FUNCTION_BLOCK PUBLIC FINAL FB_CodedOutputStream
VAR_IN_OUT
    aBuffer : ARRAY [*] OF BYTE;
END_VAR
VAR
    stState : ST_WriterInternalState;
END_VAR

{warning 'TODO: Field codecs for FB_CodedOutputStream'}
VAR
//     fbFieldCodecInt32           : FB_FieldCodecInt32;
    fbFieldCodecUInt32          : FB_FieldCodecUInt32;
//     fbFieldCodecInt64       : FB_FieldCodecInt64;
//     fbFieldCodecSInt32      : FB_FieldCodecSInt32;
//     fbFieldCodecSInt64      : FB_FieldCodecSInt64;
//     fbFieldCodecFixed32     : FB_FieldCodecFixed32;
//     fbFieldCodecFixed64     : FB_FieldCodecFixed64;    
//     fbFieldCodecFloat       : FB_FieldCodecFloat;
//     fbFieldCodecDouble      : FB_FieldCodecDouble;
    fbFieldCodecString      : FB_FieldCodecString;
//     fbFieldCodecBytes       : FB_FieldCodecBytes;
//     fbFieldCodecBool        : FB_FieldCodecBool;
END_VAR

METHOD PUBLIC FromBuffer : HRESULT
VAR
    hr : HRESULT;
END_VAR

Reset();

hr := ValidateBuffer(aBuffer);
IF FAILED(hr) THEN
    FromBuffer := hr;
    RETURN;
END_IF

Init(aBuffer);
END_METHOD

METHOD PRIVATE Init
VAR_IN_OUT CONSTANT
    aBuffer : ARRAY [*] OF BYTE;
END_VAR
VAR
    nSize : DINT;
END_VAR

stState.nBufferPos := TO_UDINT(LOWER_BOUND(aBuffer, 1));

nSize := UPPER_BOUND(aBuffer, 1) - LOWER_BOUND(aBuffer, 1);
stState.nBufferSize := TO_UDINT(nSize);
END_METHOD

PROPERTY nSpaceLeft : UDINT
GET
nSpaceLeft := stState.nBufferSize - stState.nBufferPos;
END_GET
END_PROPERTY

METHOD PRIVATE Reset
VAR_INPUT
END_VAR

stState.bError := FALSE;
stState.eWriterErrorCode := S_OK;
stState.nBufferPos := 0;
stState.nBufferSize := 0;
END_METHOD

METHOD PRIVATE ValidateBuffer : HRESULT
VAR_IN_OUT CONSTANT
    aBuffer : ARRAY[*] OF BYTE;
END_VAR
VAR
    nSize : DINT;
END_VAR
IF LOWER_BOUND(aBuffer, 1) < 0 THEN
    ValidateBuffer := E_CodedOutputStreamErrorCode.BUFFER_LOWER_BOUND;
    RETURN;
END_IF

nSize := UPPER_BOUND(aBuffer, 1) - LOWER_BOUND(aBuffer, 1);
IF nSize = 0 OR TO_UDINT(nSize) >  Param_PB.cMaxProtobufRawBuffer THEN
    ValidateBuffer := E_CodedOutputStreamErrorCode.BUFFER_SIZE;
    RETURN;
END_IF
END_METHOD

METHOD WriteBool : HRESULT
VAR_INPUT
    bValue : BOOL;
END_VAR

WriteBool := F_WriteRawByte(aBuffer, stState, TO_BYTE(bValue));
END_METHOD

METHOD WriteBytes : HRESULT
VAR_IN_OUT CONSTANT
    aBytes  : ARRAY [*] OF BYTE;
END_VAR
VAR_INPUT
    nLength : UDINT;
END_VAR

WriteBytes := F_WriteBytes(aBuffer, stState, aBytes, nLength);
END_METHOD

METHOD WriteDouble : HRESULT
VAR_INPUT
    fValue : LREAL;
END_VAR
WriteDouble := F_WriteDouble(aBuffer, stState, fValue);
END_METHOD

METHOD WriteEnum : HRESULT
VAR_INPUT
    nValue : DINT;
END_VAR

WriteEnum := F_WriteEnum(aBuffer, stState, nValue);
END_METHOD

METHOD WriteFixed32 : HRESULT
VAR_INPUT
    nValue : UDINT;
END_VAR

WriteFixed32 := F_WriteFixed32(aBuffer, stState, nValue);
END_METHOD

METHOD WriteFixed64 : HRESULT
VAR_INPUT
    nValue : ULINT;
END_VAR

WriteFixed64 := F_WriteFixed64(aBuffer, stState, nValue);
END_METHOD

METHOD WriteFloat : HRESULT
VAR_INPUT
    fValue : REAL;
END_VAR
WriteFloat := F_WriteFloat(aBuffer, stState, fValue);
END_METHOD

METHOD WriteInt32 : HRESULT
VAR_INPUT
    nValue : DINT;
END_VAR
WriteInt32 := F_WriteInt32(aBuffer, stState, nValue);
END_METHOD

METHOD WriteInt64 : HRESULT
VAR_INPUT
    nValue : LINT;
END_VAR
WriteInt64 := F_WriteInt64(aBuffer, stState, nValue);
END_METHOD

METHOD WriteLength : HRESULT
VAR_INPUT
    nLength : UDINT;
END_VAR

WriteLength := F_WriteLength(aBuffer, stState, nLength);
END_METHOD

METHOD WriteRepeatedFieldString : HRESULT
VAR_INPUT CONSTANT
    anyArray        : T_Any;
    anyFirstElem    : T_Any; 
    nLength         : UDINT;
    nTag            : UDINT;
END_VAR

WriteRepeatedFieldString := F_WriteRepeatedField(aBuffer, stState, anyArray, anyFirstElem, nLength, nTag, THIS^.fbFieldCodecString);
END_METHOD

METHOD WriteRepeatedFieldUInt32 : HRESULT
VAR_INPUT CONSTANT
    anyArray        : T_Any;
    anyFirstElem    : T_Any; 
    nLength         : UDINT;
    nTag            : UDINT;
END_VAR


WriteRepeatedFieldUInt32 := F_WriteRepeatedField(aBuffer, stState, anyArray, anyFirstElem, nLength, nTag, THIS^.fbFieldCodecUInt32);
END_METHOD

METHOD WriteSFixed32 : HRESULT
VAR_INPUT
    nValue : DINT;
END_VAR

WriteSFixed32 := F_WriteSFixed32(aBuffer, stState, nValue);
END_METHOD

METHOD WriteSFixed64 : HRESULT
VAR_INPUT
    nValue : LINT;
END_VAR

WriteSFixed64 := F_WriteSFixed64(aBuffer, stState, nValue);
END_METHOD

METHOD WriteSint32 : HRESULT
VAR_INPUT
    nValue : DINT;
END_VAR
WriteSint32 := F_WriteSInt32(aBuffer, stState, nValue);
END_METHOD

METHOD WriteSint64 : HRESULT
VAR_INPUT
    nValue : LINT;
END_VAR
WriteSint64 := F_WriteSInt64(aBuffer, stState, nValue);
END_METHOD

METHOD WriteString : HRESULT
VAR_IN_OUT CONSTANT
    sStringToWrite          : T_ProtobufMaxString;
END_VAR

WriteString := F_WriteString(aBuffer, stState, sStringToWrite);
END_METHOD

METHOD WriteTag : HRESULT
VAR_INPUT
    nFieldNumber    : UDINT;
    eWireType       : E_WireType;
END_VAR

WriteTag := F_WriteTag(aBuffer, stState, nFieldNumber, eWireType);
END_METHOD

METHOD WriteUint32 : HRESULT
VAR_INPUT
    nValue : UDINT;
END_VAR


WriteUint32 := F_WriteUInt32(aBuffer, stState, nValue);
END_METHOD

METHOD WriteUint64 : HRESULT
VAR_INPUT
    nValue : ULINT;
END_VAR
WriteUint64 := F_WriteUInt64(aBuffer, stState, nValue);
END_METHOD

END_FUNCTION_BLOCK

(* stored: Version 1.1.0.1
   POU FB_CodedOutputStream: Id {18246595-6bbb-43ef-aa75-24f9e22ace2b}, SpecialFunc None
   Method FromBuffer: Id {c2539802-bec0-4365-8257-fc8ef3ad282b}
   Method Init: Id {a9471daf-b84d-4c35-956f-348eed5a15a5}
   Property nSpaceLeft: Id {81be7da9-2e5d-48e4-88e3-0f185cdb7127}
   Get Get: Id {060dd1c8-d1ad-424e-8a91-006db807548b}
   Method Reset: Id {7023c71a-5838-4abb-a6b6-612b36e632a1}
   Method ValidateBuffer: Id {64be83e4-6577-460a-b1a5-dcd5db2f4e92}
   Method WriteBool: Id {959509b8-b6ba-41cc-a129-8f0ea33bc2ff}
   Method WriteBytes: Id {02b8f0af-661f-4944-85ff-f76fd4cec3ea}
   Method WriteDouble: Id {3b86ec3f-2cad-45c5-9a6f-d56de79d1415}
   Method WriteEnum: Id {4fb9d4ab-4be6-42ee-a3bb-3f86dbf2061c}
   Method WriteFixed32: Id {75c23fcd-723d-4cbc-9e77-8e2301b57ac1}
   Method WriteFixed64: Id {ac5b07e1-2d27-4aea-84db-e2a22552a9fb}
   Method WriteFloat: Id {ec5060f6-e490-4798-a185-1d013ad3518c}
   Method WriteInt32: Id {cb424f8c-2286-402b-adff-21634a582503}
   Method WriteInt64: Id {470d349f-a883-451f-86ff-5add09c6bbc1}
   Method WriteLength: Id {aefabf76-233a-48e5-bd46-c3bd214198fb}
   Method WriteRepeatedFieldString: Id {3c1dcc4b-c34b-4c95-a10d-fb1de4f1751e}
   Method WriteRepeatedFieldUInt32: Id {7d0ba148-7c14-4624-856c-284819f70ded}
   Method WriteSFixed32: Id {c5db7557-6b1a-4521-ab52-97e9e0d0670f}
   Method WriteSFixed64: Id {1d1909aa-43d1-452a-93e7-9bb5567d60cd}
   Method WriteSint32: Id {9b3c1ae8-a598-4a54-9dcf-fc39ef583879}
   Method WriteSint64: Id {b35dcafc-ac19-4012-a560-388617eee3d1}
   Method WriteString: Id {e0704046-198b-43d6-993d-44c5595830da}
   Method WriteTag: Id {7d0d5de0-234e-4fd9-b783-7b62ad087c0a}
   Method WriteUint32: Id {5d55f154-a20b-441b-9140-093b322d95f5}
   Method WriteUint64: Id {340b2f1b-3da7-48bf-82ca-67d4a8315258} *)
